// Mitsubishi GX Works2 project: FrekvensMLDEdit   PLC: FX1S

// global labels: Global1
VAR_GLOBAL
  Sens_1 AT X002 : BOOL;
  Sens_2 AT X003 : BOOL;
  Sens_3 AT X004 : BOOL;
  Sens_4 AT X005 : BOOL;
  Start AT X000 : BOOL;
  Reset AT X001 : BOOL;
  Stage_1 AT M0 : BOOL;
  Stage_2 AT M1 : BOOL;
  Stage_3 AT M2 : BOOL;
  Stage_4 AT M3 : BOOL;
  Stage_5 AT M4 : BOOL;
  Stage_6 AT M5 : BOOL;
  Stage_7 AT M6 : BOOL;
  Forward AT Y000 : BOOL;
  Back AT Y001 : BOOL;
  F1 AT Y003 : BOOL;
  F2 AT Y002 : BOOL;
  F3 AT Y004 : BOOL;
END_VAR

// task Task_01 (event TRUE, interval 0, priority 31): Sequence, Activation

PROGRAM Sequence
VAR
  Run : BOOL;
  Seq_Ct : CTU;
  Timer_In : TON;
  StartDelay : TON;
  Timer_Out : TON;
END_VAR
(* structured ladder/FBD written out as ST: instructions are called as NAME(EN, inputs, outputs); _pN, _eN, _tN stand for wires *)
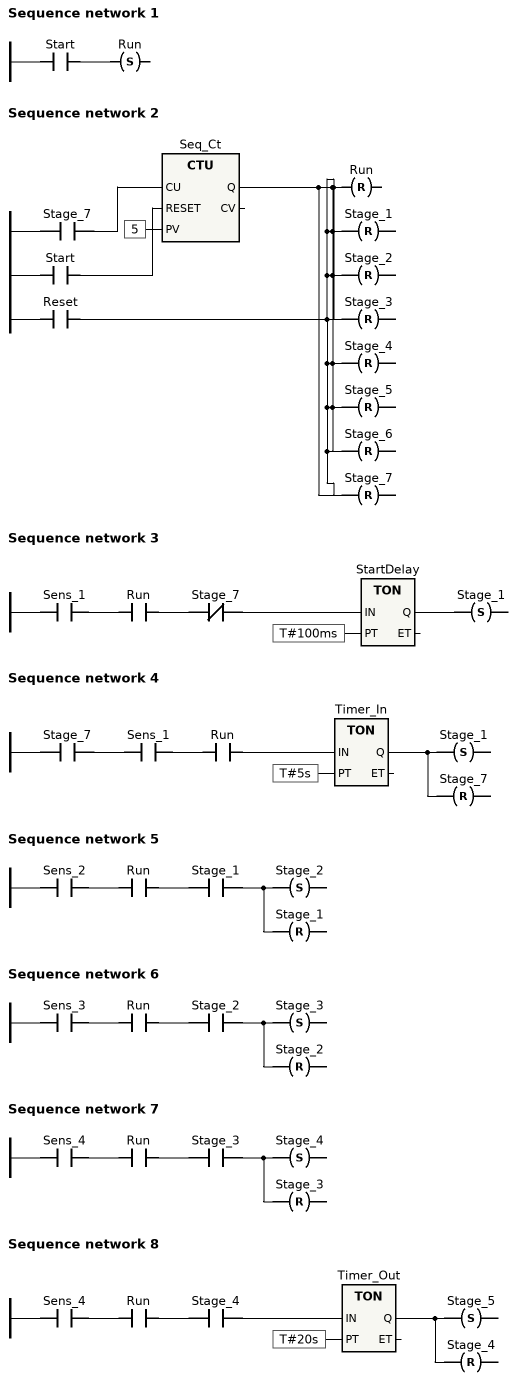
(* network 1 *)
SET(Start, Run);
(* network 2 *)
Seq_Ct(CU := Stage_7, RESET := Start, PV := 5);
_p1 := Seq_Ct.Q OR Reset;
RST(_p1, Run);
RST(_p1, Stage_1);
RST(_p1, Stage_2);
RST(_p1, Stage_3);
RST(_p1, Stage_4);
RST(_p1, Stage_5);
RST(_p1, Stage_6);
RST(_p1, Stage_7);
(* network 3 *)
StartDelay(IN := Sens_1 AND Run AND NOT Stage_7, PT := T#100ms);
SET(StartDelay.Q, Stage_1);
(* network 4 *)
Timer_In(IN := Stage_7 AND Sens_1 AND Run, PT := T#5s);
SET(Timer_In.Q, Stage_1);
RST(Timer_In.Q, Stage_7);
(* network 5 *)
_p1 := Sens_2 AND Run AND Stage_1;
SET(_p1, Stage_2);
RST(_p1, Stage_1);
(* network 6 *)
_p1 := Sens_3 AND Run AND Stage_2;
SET(_p1, Stage_3);
RST(_p1, Stage_2);
(* network 7 *)
_p1 := Sens_4 AND Run AND Stage_3;
SET(_p1, Stage_4);
RST(_p1, Stage_3);
(* network 8 *)
Timer_Out(IN := Sens_4 AND Run AND Stage_4, PT := T#20s);
SET(Timer_Out.Q, Stage_5);
RST(Timer_Out.Q, Stage_4);
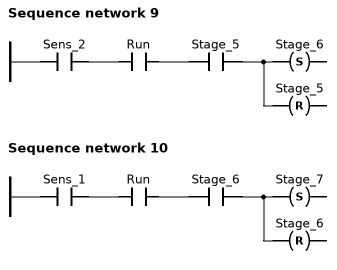
(* network 9 *)
_p1 := Sens_2 AND Run AND Stage_5;
SET(_p1, Stage_6);
RST(_p1, Stage_5);
(* network 10 *)
_p1 := Sens_1 AND Run AND Stage_6;
SET(_p1, Stage_7);
RST(_p1, Stage_6);
END_PROGRAM

PROGRAM Activation
VAR
  Timer_Out : TON;
  FMinne2 : BOOL;
  FMinne3 : BOOL;
  FMinne1 : BOOL;
END_VAR
(* structured ladder/FBD written out as ST: instructions are called as NAME(EN, inputs, outputs); _pN, _eN, _tN stand for wires *)
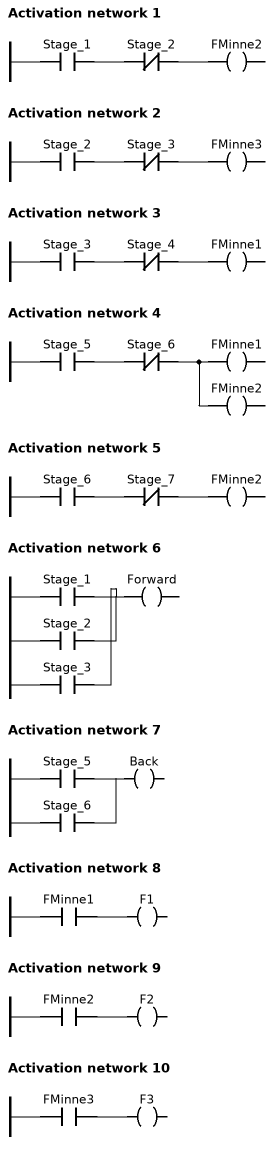
(* network 1 *)
FMinne2 := Stage_1 AND NOT Stage_2;
(* network 2 *)
FMinne3 := Stage_2 AND NOT Stage_3;
(* network 3 *)
FMinne1 := Stage_3 AND NOT Stage_4;
(* network 4 *)
_p1 := Stage_5 AND NOT Stage_6;
FMinne1 := _p1;
FMinne2 := _p1;
(* network 5 *)
FMinne2 := Stage_6 AND NOT Stage_7;
(* network 6 *)
Forward := Stage_1 OR Stage_2 OR Stage_3;
(* network 7 *)
Back := Stage_5 OR Stage_6;
(* network 8 *)
F1 := FMinne1;
(* network 9 *)
F2 := FMinne2;
(* network 10 *)
F3 := FMinne3;
END_PROGRAM
